FUNCTION_BLOCK AxisControl
VAR_INPUT
	Axis 			: AXIS_REF;
	AxisInputs		: AxisInputs;
END_VAR
VAR_OUTPUT
	Status			: AxisFeedback;
END_VAR
VAR
	Power			: MC_Power;
	Reset			: MC_Reset;
	Stop			: MC_Stop;
	Jog				: MC_Jog;
	Halt			: MC_Halt;
	MoveAbsolute	: MC_MoveAbsolute;
	MoveRelative	: MC_MoveRelative;
END_VAR

Power(Axis := Axis,
	  Enable := AxisInputs.PowerEnable,
	  Enable_Positive := AxisInputs.EnablePositive,
	  Enable_Negative := AxisInputs.EnableNegative,
	  Override := AxisInputs.Override,
	  BufferMode := AxisInputs.BufferMode,
	  Options := AxisInputs.Options,
	  Status => Status.Status,
	  Busy => Status.Busy,
	  Active => Status.Active,
	  Error => Status.Error,
	  ErrorID => Status.ErrorID);

	 
Reset(Axis := Axis,
	  Execute := AxisInputs.ResetEnable,
	  Done => Status.Done,
      Busy => Status.Busy,
	  Error => Status.Busy,
	  ErrorID => Status.ErrorID);
	  
Stop(Axis := Axis,
	 Execute := AxisInputs.StopExecute,
	 Deceleration := AxisInputs.StopDeceleration,
	 Jerk := AxisInputs.StopJerk,
	 Options := AxisInputs.StopOptions,
	 Done => Status.Done,
	 Busy => Status.Busy,
	 Active => Status.Active,
	 CommandAborted => Status.CommandAborted,
	 Error => Status.Error,
	 ErrorID => Status.ErrorID); 

Halt(Axis := Axis,
	 Execute := AxisInputs.HaltExecute,
	 Deceleration := AxisInputs.HaltDeceleration,
	 Jerk := AxisInputs.HaltJerk,
	 BufferMode := AxisInputs.HaltBufferMode,
	 Options := AxisInputs.HaltOptions,
	 Done => Status.Done,
	 Busy => Status.Busy,
	 Active => Status.Active,
	 CommandAborted => Status.CommandAborted,
	 Error => Status.Error,
	 ErrorID => Status.ErrorID); 

Jog(Axis := Axis,
	JogForward := AxisInputs.JogForward,
	JogBackwards := AxisInputs.JogBackward,
	Mode := AxisInputs.jogMode,
	Position := AxisInputs.JogPosition,
	Velocity := AxisInputs.JogVelocity,
	Acceleration := AxisInputs.JogAcceleration,
	Deceleration := AxisInputs.JogDeceleration,
	jerk := AxisInputs.JogJerk,
	Done => Status.Done,
	Busy => Status.Busy,
	Active => Status.Active,
	CommandAborted => Status.CommandAborted,
	Error => Status.Error,
	ErrorID => Status.ErrorID);
	
MoveAbsolute(Axis := Axis,
			 Execute := AxisInputs.MoveAbsoluteExecute,
			 Position := AxisInputs.MoveAbsolutePosition,
			 Acceleration := AxisInputs.MoveAbsoluteAcceleration,
			 Deceleration := AxisInputs.MoveAbsoluteDeceleration,
			 Jerk := AxisInputs.MoveAbsoluteJerk,
			 Options := AxisInputs.MoveAbsoluteOptions,
			 BufferMode := AxisInputs.MoveAbsoluteBufferMode,
			 Done => Status.Done,
			 Busy => Status.Busy,
			 Active => Status.Active,
			 CommandAborted => Status.CommandAborted,
			 Error => Status.Error,
			 ErrorID => Status.ErrorID);
				 
MoveRelative(Axis := Axis,
			 Execute := AxisInputs.MoveRelativeExecute,
			 Distance := AxisInputs.MoveRelativeDistance,
			 Acceleration := AxisInputs.MoveRelativeAcceleration,
			 Deceleration := AxisInputs.MoveRelativeDeceleration,
			 Jerk := AxisInputs.MoveRelativeJerk,
			 Options := AxisInputs.MoveRelativeOptions,
			 BufferMode := AxisInputs.MoveRelativeBufferMode,
			 Done => Status.Done,
			 Busy => Status.Busy,
			 Active => Status.Active,
			 CommandAborted => Status.CommandAborted,
			 Error => Status.Error,
			 ErrorID => Status.ErrorID);

END_FUNCTION_BLOCK

(* stored: Version 1.1.0.1, ProductVersion 3.1.4024.10
   POU AxisControl: Id {9f87289e-6749-4cbb-bb3a-569f3c84f8a5}, SpecialFunc None *)
